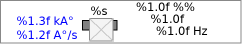
VISUALIZATION VISU_XTAL  // 242x44
VAR_IN_OUT
	m_Input_XTAL : BLOCK_XTAL;
END_VAR
    Rectangle (1,14 85x14), "%1.3f kA°", text variable: m_Input_XTAL.STATE_THICKNESS
    Rectangle (81,3 36x16), "%s", text variable: m_Input_XTAL.MNEMO
    Rectangle (82,20 35x10)
    RoundedRectangle (92,28 17x7)
    Rectangle (121,0 86x14), "%1.0f %%", text variable: m_Input_XTAL.STATE_Life
    Rectangle (120,24 120x14), "%1.0f Hz", text variable: m_Input_XTAL.STATE_FREQUENCY
    Rectangle (121,12 89x14), "%1.0f", text variable: m_Input_XTAL.STATE_ACTIVITY
    Rectangle (3,28 85x14), "%1.2f A°/s", text variable: m_Input_XTAL.STATE_RATE
    Image (89,18 24x23), invisible if: NOT m_Input_XTAL.STATE_NOK, image: MesImages.warning
END_VISUALIZATION

(* stored: Version 1.1.0.1, ProductVersion 3.1.4024.10
   Visu VISU_XTAL: Id {dcd1ce66-cfa8-4f5e-ae5a-5e0024c3dd6d} *)
